FUNCTION Mapping_Monitoring_Variables_ABG
VAR_INPUT
	Input_var : ModbusRead;//ScaledModRead;
	Output_var : POINTER TO EtherCAT_Monitor_Variables;
	Output_var2 : POINTER TO EtherCAT_Stat_Variables;
END_VAR
VAR
END_VAR

Output_var^.BatSoc := (Input_var.BatSoc );
Output_var^.BatSocLowLim := (Input_var.BatSocLowLim);
Output_var^.BatSocUpLim := (Input_var.BatSocUpLim );

CASE Input_var.DerOpMode	OF
	0:	
		Output_var2^.Status := 0;
	1:	
		Output_var2^.Status := 0;
	4:
		Output_var2^.Status := 1;
	11:
		Output_var2^.Status := 1;
	5:
		Output_var2^.Status := 2;
	6:
		Output_var2^.Status := 3;
	9:
		Output_var2^.Status := 5;
END_CASE

//Output_var2^.Status := Input_var.DerOpMode;


Output_var2^.HeartBeat := GlobalVar.wMiliseconds;

Output_var2^.Alarms1 := UDINT_TO_DINT((Input_var.GrAlm));
Output_var2^.Alarms2 := 0; //Input_var.GrAlm1;
Output_var2^.Alarms3 := 0; //Input_var.GrAlm2;
Output_var2^.Alarms4 := 0; //Input_var.GrAlm3;

Output_var^.GridFre := (Input_var.GridFre);

Output_var^.Irmsa := (Input_var.Irmsa);
Output_var^.Irmsb := (Input_var.Irmsb);
Output_var^.Irmsc := (Input_var.Irmsc);

Output_var^.TotW := (Input_var.TotW);
Output_var^.TotVAr := (Input_var.TotVAr);

Output_var^.Vrmsa := (Input_var.Vrmsa);
Output_var^.Vrmsb := (Input_var.Vrmsb);
Output_var^.Vrmsc := (Input_var.Vrmsc);

END_FUNCTION

(* stored: Version 1.1.0.1, ProductVersion 3.1.4024.4
   POU Mapping_Monitoring_Variables_ABG: Id {acb49f2e-cde5-4859-a7e0-79f191ed30c3}, SpecialFunc None *)
